// TIA Portal V19 export
DATA_BLOCK "EnS_Buffer32469"   // DB2
TITLE = Global DB for buffer data
AUTHOR : Siemens
FAMILY : EnS
// Global DB for buffer data
   STRUCT
      EnS_Buffer32469 : Array[0..114] of "EnS_typeValue";
   END_STRUCT;
BEGIN
END_DATA_BLOCK
